FUNCTION_BLOCK Empty
  (* Version 1.0, 2007-10-25, Goran Cengic, Chalmers *)
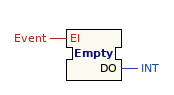
  EVENT_INPUT
    EI;
  END_EVENT
  VAR_OUTPUT
    DO : INT;
  END_VAR
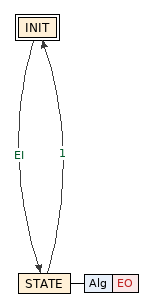
  EC_STATES
    INIT;
    STATE : Alg -> EO;
  END_STATES
  EC_TRANSITIONS
    INIT TO STATE := EI;
    STATE TO INIT := 1;
  END_TRANSITIONS
  ALGORITHM Alg IN Java:
		DO = 1;
  END_ALGORITHM
END_FUNCTION_BLOCK
(* other elements stored in the file *)
(* Event Name=EO *)
(* With Var=DO *)
